# EPICS IOC start-up script: iocsh/ethercatmcMotorTemp.iocsh
ethercatmcCreateAsynParam $(MOTOR_PORT) MotorTemp Float64

dbLoadRecords("ethercatmcMotorTemp.template", "P=$(P), R=$(R), DESC=$(DESC), MOTOR_PORT=$(MOTOR_PORT), AXIS_NO=$(AXIS_NO)")
